PROGRAM MAIN
VAR
END_VAR

PRG_Mainprg();
PRG_CONTROLM1();

FIO_Read_Inputs();
FIO_Write_Outputs();
ReadWriteIO();

END_PROGRAM

(* stored: Version 1.1.0.1
   POU MAIN: Id {1fc035af-53d0-4100-abf7-dbd437ade9fb}, SpecialFunc None *)
